SYSTEM FLASHER_TEST (* Flasher Test System Configuration *)
  (* Standard: 61499-1 *)
  (* Version 0.0, 2001-07-31, JHC, Rockwell Automation, Changed IN_TIME to IN_ANY, adjusted height. *)
  (* Version 0.0, 2001-02-22, JHC, Rockwell Automation *)
  DEVICE FLASHER : FRAME_DEVICE
    RESOURCE RES1 : PANEL_RESOURCE
      FBS
        START_PB : IN_EVENT;
        STOP_PB : IN_EVENT;
        DT : IN_ANY;
        PERIODIC : E_CYCLE;
        MODE : IN_CHOICE;
        FLASHIT : FLASHER4;
        LEDS : LED_HMI;
      END_FBS
      EVENT_CONNECTIONS
        START.COLD TO START_PB.INIT;
        START_PB.INITO TO STOP_PB.INIT;
        STOP_PB.INITO TO DT.INIT;
        DT.INITO TO MODE.INIT;
        MODE.INITO TO FLASHIT.INIT;
        FLASHIT.INITO TO LEDS.INIT;
        START_PB.IND TO DT.REQ;
        DT.IND TO PERIODIC.START;
        STOP_PB.IND TO PERIODIC.STOP;
        MODE.IND TO FLASHIT.INIT;
        PERIODIC.EO TO FLASHIT.REQ;
        FLASHIT.CNF TO LEDS.REQ;
      END_CONNECTIONS
      DATA_CONNECTIONS
        DT.OUT TO PERIODIC.DT;
        1 TO MODE.QI;
        MODE.I TO FLASHIT.MODE;
        FLASHIT.LED3 TO LEDS.LED3;
        FLASHIT.LED2 TO LEDS.LED2;
        FLASHIT.LED1 TO LEDS.LED1;
        FLASHIT.LED0 TO LEDS.LED0;
        "FLASH_ALL,COUNT_UP,COUNT_DOWN,CHASE_UP,CHASE_DOWN" TO MODE.CHOICES;
        1 TO START_PB.QI;
        1 TO STOP_PB.QI;
        "START" TO START_PB.LABEL;
        "STOP" TO STOP_PB.LABEL;
        1 TO DT.QI;
        "TIME" TO DT.TYPE;
        t#250ms TO DT.IVAL;
      END_CONNECTIONS
    END_RESOURCE
    DATA_CONNECTIONS
      0 TO RES1.TRACE;
    END_CONNECTIONS
  END_DEVICE
  DATA_CONNECTIONS (* parameter values *)
    [100,100,320,100] TO FLASHER.BOUNDS;
    [1,1] TO FLASHER.GRID;
  END_CONNECTIONS
END_SYSTEM
